(* CODESYS project Abstract Factory2.project

Project tree, tasks and I/O mapping:
  Device : CODESYS Control for Raspberry Pi SL, 3S - Smart Software Solutions GmbH, version 3.5.11.0
    application Application
      libraries: Standard, * (System); StringUtils, 3.5.11.0 (System); CoDeSys Memory Manager, 3.5.12.0 (3S - Smart Software Solutions GmbH)
      task Task (cyclic, interval t#20ms, priority 1) calls MAIN
      POUs/
        function block FB_FileLoggerFactory [ST]: FB_init, GetLogger, FB_exit
        function block FB_Logger [ST]: Write, FB_init
        function block FB_TxtLogger [ST]: Write
        function block FB_CsvLogger [ST]: Write
        function block FB_XmlLogger [ST]: Write
        function block FB_AbstractLoggerFactory [ST]: GetLogger
        interface ILogger: Write
        program MAIN [ST]
    SoftMotion General Axis Pool
    I²C
    SPI
    GPIOs_A_B : GPIOs A/B, 3S - Smart Software Solutions GmbH, version 3.5.11.0
        unmapped channels: digital inputs (GPIO0..GPIO31), digital outputs (GPIO0..GPIO31)
    Onewire
    Camera device
      <Empty>
*)

// Device/Application/POUs/MAIN
PROGRAM MAIN
VAR
	fbFileLoggerFactory	  : FB_FileLoggerFactory('File.csv');
	refFileLoggerFactory  : REFERENCE TO FB_FileLoggerFactory := fbFileLoggerFactory;
	fbLogger 			  : FB_Logger(refFileLoggerFactory);	
	sRetMsg				  : STRING;
END_VAR

sRetMsg := fbLogger.Write('Hello');

END_PROGRAM

// Device/Application/POUs/FB_FileLoggerFactory
FUNCTION_BLOCK INTERNAL FB_FileLoggerFactory EXTENDS FB_AbstractLoggerFactory
VAR
	pTxtLogger  : POINTER TO FB_TxtLogger;
	pCsvLogger  : POINTER TO FB_CsvLogger;
	pXmlLogger  : POINTER TO FB_XmlLogger;
    ipLogger    : ILogger := 0;
END_VAR

METHOD FB_init : BOOL
VAR_INPUT
    bInitRetains  : BOOL; // if TRUE, the retain variables are initialized (warm start / cold start)
    bInCopyCode   : BOOL;  // if TRUE, the instance afterwards gets moved into the copy code (online change)
    sFilename     : STRING;
END_VAR
VAR
    sFilenameExtension : STRING;
END_VAR
sFilenameExtension := RIGHT(sFilename, 3);
IF (sFilenameExtension = 'txt' OR sFilenameExtension = 'TXT') THEN
    pTxtLogger := __NEW(FB_TxtLogger);
    ipLogger := pTxtLogger^;
ELSIF (sFilenameExtension = 'csv' OR sFilenameExtension = 'CSV') THEN
    pCsvLogger := __NEW(FB_CsvLogger);
    ipLogger := pCsvLogger^;
ELSIF (sFilenameExtension = 'xml' OR sFilenameExtension = 'XML') THEN
    pXmlLogger := __NEW(FB_XmlLogger);
    ipLogger := pXmlLogger^;
ELSE
    ipLogger := 0;
END_IF
END_METHOD

METHOD PUBLIC GetLogger : ILogger
VAR_INPUT
END_VAR
GetLogger := ipLogger;
END_METHOD

METHOD FB_exit : BOOL
VAR_INPUT
	bInCopyCode : BOOL; // if TRUE, the exit method is called for exiting an instance that is copied afterwards (online change).
END_VAR
IF (pTxtLogger <> 0) THEN
	__DELETE(pTxtLogger);
	pTxtLogger := 0;
END_IF

IF (pCsvLogger <> 0) THEN
	__DELETE(pCsvLogger);
	pCsvLogger := 0;
END_IF

IF (pXmlLogger <> 0) THEN
	__DELETE(pXmlLogger);
	pXmlLogger := 0;
END_IF
END_METHOD

END_FUNCTION_BLOCK

// Device/Application/POUs/FB_AbstractLoggerFactory
FUNCTION_BLOCK public FB_AbstractLoggerFactory
VAR_INPUT
END_VAR
VAR_OUTPUT
END_VAR
VAR
END_VAR

METHOD PUBLIC GetLogger : ILogger
VAR_INPUT
END_VAR
;
END_METHOD

END_FUNCTION_BLOCK

// Device/Application/POUs/ILogger
INTERFACE ILogger

METHOD Write : STRING
VAR_INPUT
	sMsg	: STRING;
END_VAR
END_METHOD

END_INTERFACE

// Device/Application/POUs/FB_TxtLogger
{attribute 'enable_dynamic_creation'}
FUNCTION_BLOCK INTERNAL FB_TxtLogger IMPLEMENTS ILogger
VAR_INPUT
END_VAR
VAR_OUTPUT
END_VAR
VAR
END_VAR

METHOD PUBLIC Write : STRING
VAR_INPUT
	sMsg : STRING;
END_VAR
Write := CONCAT('TxtLogger: ', sMsg);
END_METHOD

END_FUNCTION_BLOCK

// Device/Application/POUs/FB_CsvLogger
{attribute 'enable_dynamic_creation'}
FUNCTION_BLOCK INTERNAL FB_CsvLogger IMPLEMENTS ILogger
VAR_INPUT
END_VAR
VAR_OUTPUT
END_VAR
VAR
END_VAR

METHOD PUBLIC Write : STRING
VAR_INPUT
	sMsg : string;
END_VAR
Write := CONCAT('CsvLogger: ', sMsg);
END_METHOD

END_FUNCTION_BLOCK

// Device/Application/POUs/FB_XmlLogger
{attribute 'enable_dynamic_creation'}
FUNCTION_BLOCK INTERNAL FB_XmlLogger IMPLEMENTS ILogger
VAR_INPUT
END_VAR
VAR_OUTPUT
END_VAR
VAR
END_VAR

METHOD PUBLIC Write : STRING
VAR_INPUT
	sMsg	: string;
END_VAR
Write := CONCAT('XmlLogger: ', sMsg);
END_METHOD

END_FUNCTION_BLOCK

// Device/Application/POUs/FB_Logger
FUNCTION_BLOCK PUBLIC FB_Logger
VAR
	ipLogger : ILogger;
END_VAR

METHOD PUBLIC Write : STRING
VAR_INPUT
	sMsg 		 : STRING;
END_VAR
Write := 'Error';
IF (ipLogger <> 0) THEN
	Write := ipLogger.Write(sMsg);
END_IF
END_METHOD

METHOD FB_init : BOOL
VAR_INPUT
	bInitRetains       : BOOL; // if TRUE, the retain variables are initialized (warm start / cold start)
	bInCopyCode        : BOOL;  // if TRUE, the instance afterwards gets moved into the copy code (online change)
	refLoggerFactory   : REFERENCE TO FB_AbstractLoggerFactory;
END_VAR
IF (__ISVALIDREF(refLoggerFactory)) THEN
	ipLogger := refLoggerFactory.GetLogger();
ELSE
	ipLogger := 0;
END_IF
END_METHOD

END_FUNCTION_BLOCK
